SUBAPPLICATION Ventilsteuerung_Uebung_002c (* DigitalInput_I1 auf DigitalOutput_Q1 *)
  (* Standard: 61499-2 *)
  (* Version 1.0, 2023-10-23, franz *)
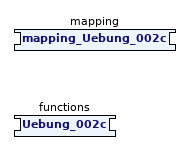
  SUBAPPS
    mapping : mapping_Uebung_002c;
    functions : Uebung_002c;
  END_SUBAPPS
END_SUBAPPLICATION
